// TIA Portal V20 export
VAR_GLOBAL   // PLC tag table "Default tag table"
   dfsq AT %I0.1 : Bool;
END_VAR
